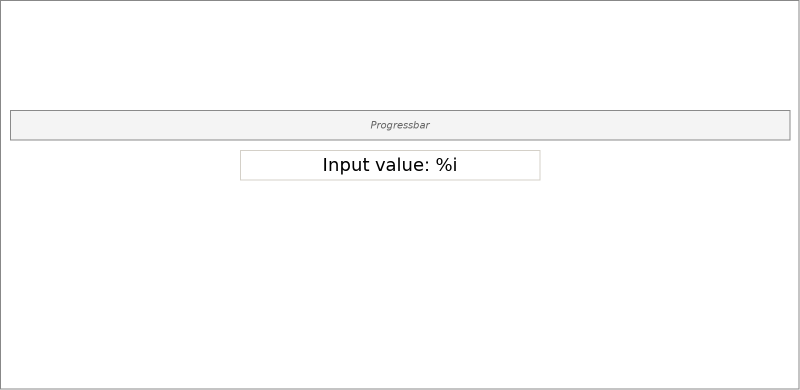
VISUALIZATION VisuAnlogInputControl  // 800x390
VAR_IN_OUT
	fbManualControler	: FB_ManualController ;
END_VAR
    Progressbar (10,110 780x30), variable: fbManualControler.pDevAnalogInput^.fValue
    Textfield (240,150 300x30), "Input value: %i", text variable: fbManualControler.pDevAnalogInput^.fValue
END_VISUALIZATION

(* stored: Version 1.1.0.1, ProductVersion 3.1.4024.9
   Visu VisuAnlogInputControl: Id {05161f7c-ba6d-4f2f-9bcb-245dad7521da} *)
